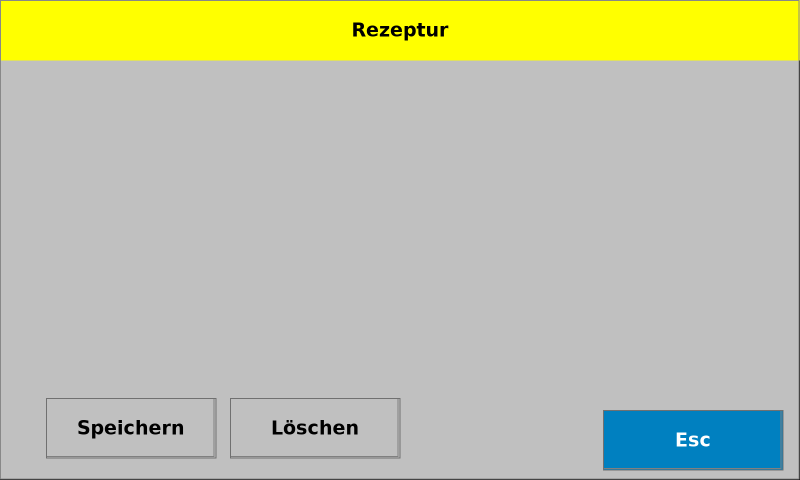
VISUALIZATION Rezeptur  // 800x480
    Rectangle (0,0 800x480)
    Rectangle (0,0 800x60), "Rezeptur"
    Button (603,410 180x60), "Esc"
        OnMouseUp: change screen: Previous 
    Button (46,398 170x60), "Speichern"
    Button (230,398 170x60), "Löschen"
END_VISUALIZATION

(* stored: Version 1.1.0.1, ProductVersion 3.1.4024.3
   Visu Rezeptur: Id {98feb544-8c65-4f6f-a4c8-cce6f7e4eb3f} *)
